Staubli VAL3: findPos.pgx

public program findPos(string x_sItem1, string x_sItem2, num& x_nPos[])
  local num l_nPos
begin
  // find the char using getDisplayLen
  l_nPos=find(x_sItem1,x_sItem2)
  if l_nPos!=-1
    x_nPos=getDisplayLen(left(x_sItem1,l_nPos))
  else
    x_nPos=-1
  endIf
end
